// TIA Portal project "PRESS1-2-3" (V18)

(* hardware
DEVICE "S7-1200 station_1"  S7-1200 Station
   slot 0: "Rack_0"  S7-1200 Rack  Rack  V1.0
   slot 1: "PLC_1"  CPU 1212C DC/DC/DC  6ES7 212-1AE40-0XB0  V4.5
*)

// ===== PLC "PLC_1"  CPU 1212C DC/DC/DC =====

VAR_GLOBAL   // PLC tag table "Tabla de variables estándar"
   "Simulem 5V (24)" AT %Q0.0 : Bool;
   "Interruptor" AT %M50.0 : Bool;
   "Off_interruptor" AT %M50.1 : Bool;
   "System_Byte" AT %MB1 : Byte;
   "FirstScan" AT %M1.0 : Bool;
   "DiagStatusUpdate" AT %M1.1 : Bool;
   "AlwaysTRUE" AT %M1.2 : Bool;
   "AlwaysFALSE" AT %M1.3 : Bool;
   "System_Byte(1)" AT %MB1 : Byte;
   "Prensa_abaix" AT %I0.0 : Bool;
   "Prensa_dalt" AT %I0.1 : Bool;
   "Selector_Automatic" AT %I0.2 : Bool;
   "Sensor_mans" AT %I0.3 : Bool;
   "Maquina_endollada" AT %I0.4 : Bool;
END_VAR

VAR_GLOBAL   // PLC tag table "senyals_okuma"
   "nova_peca" AT %I0.7 : Bool;
   "servei" AT %I0.5 : Bool;
   "pedal" AT %I0.6 : Bool;
END_VAR

DATA_BLOCK "Prensa1"   // DB2
{ S7_Optimized_Access := 'FALSE' }
VERSION : 0.1
   VAR
      num_peces : UInt;
      temps_peca : Time;
      hora_peca : DTL;
      reset : UInt;
   END_VAR
BEGIN
END_DATA_BLOCK

DATA_BLOCK "vAR_Inpas"   // DB3
{ S7_Optimized_Access := 'FALSE' }
VERSION : 0.1
   VAR
      hora_actual : DTL;
      flanc2 : Bool;
      flanc1 : Bool;
      recompte_de_peces : Array[0..300] of Time;
   END_VAR
BEGIN
END_DATA_BLOCK

FUNCTION_BLOCK "Peca_acabada"   // FB1, LAD
TITLE = obtenim: temps de peça, hora inici, hora final
{ S7_Optimized_Access := 'TRUE' }
VERSION : 0.1
   VAR RETAIN
      OPC_Data : Struct
         Data_bool : Bool;
         Data_Int : Int;
         Data_String : String;
      END_STRUCT;
   END_VAR
   VAR_TEMP
      hora_actual : DTL;
      ok : Int;
   END_VAR
BEGIN

REGION Network 1: Obtenim la hora actual (hora de peça acabada)
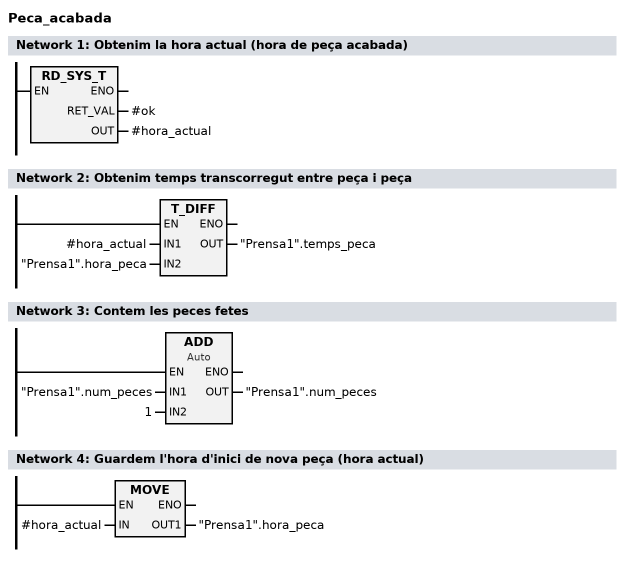
   #ok := RD_SYS_T(OUT => #hora_actual);
END_REGION

REGION Network 2: Obtenim temps transcorregut entre peça i peça
   "Prensa1".temps_peca := T_DIFF(IN1 := #hora_actual, IN2 := "Prensa1".hora_peca);
END_REGION

REGION Network 3: Contem les peces fetes
   RUNG wire#powerrail
      Add(in1 := "Prensa1".num_peces, in2 := 1, out => "Prensa1".num_peces)
   END_RUNG
   // the same network as SCL:
   "Prensa1".num_peces := "Prensa1".num_peces + 1;
END_REGION

REGION Network 4: Guardem l'hora d'inici de nova peça (hora actual)
   RUNG wire#powerrail
      Move(in := #hora_actual, out1 => "Prensa1".hora_peca)
   END_RUNG
   // the same network as SCL:
   "Prensa1".hora_peca := #hora_actual;
END_REGION
END_FUNCTION_BLOCK

FUNCTION "Peca_acabada_ok" : Void   // FC1, LAD
{ S7_Optimized_Access := 'TRUE' }
VERSION : 0.1
   VAR_INPUT
      hora_ultima_peca_in : DTL;
      num_peces_in : UInt;
   END_VAR
   VAR_OUTPUT
      hora_ultima_peca_out : DTL;
      temps_peca_out : Time;
      num_peces_out : UInt;
   END_VAR
   VAR_TEMP
      hora_actual : DTL;
      ok : Int;
   END_VAR
BEGIN

REGION Network 1: Obtenim la hora actual (hora de peça acabada)
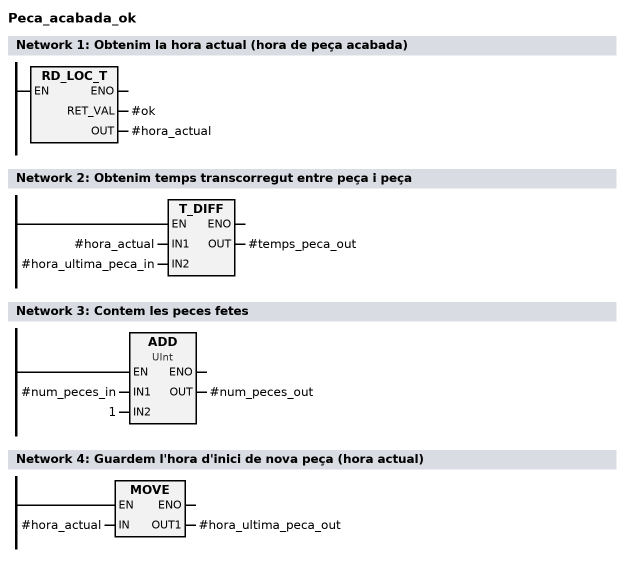
   #ok := RD_LOC_T(OUT => #hora_actual);
END_REGION

REGION Network 2: Obtenim temps transcorregut entre peça i peça
   #temps_peca_out := T_DIFF(IN1 := #hora_actual, IN2 := #hora_ultima_peca_in);
END_REGION

REGION Network 3: Contem les peces fetes
   RUNG wire#powerrail
      { S7_Templates := "SrcType := UInt" } Add(in1 := #num_peces_in, in2 := 1, out => #num_peces_out)
   END_RUNG
   // the same network as SCL:
   #num_peces_out := #num_peces_in + 1;
END_REGION

REGION Network 4: Guardem l'hora d'inici de nova peça (hora actual)
   RUNG wire#powerrail
      Move(in := #hora_actual, out1 => #hora_ultima_peca_out)
   END_RUNG
   // the same network as SCL:
   #hora_ultima_peca_out := #hora_actual;
END_REGION
END_FUNCTION

ORGANIZATION_BLOCK "Main"   // OB1, LAD, ProgramCycle
TITLE = "Main Program Sweep (Cycle)"
{ S7_Optimized_Access := 'TRUE' }
VERSION : 0.1
   VAR_INPUT
      Initial_Call : Bool;   // Initial call of this OB
      Remanence : Bool;   // =True, if remanent data are available
   END_VAR
   VAR_TEMP
      ok : Int;
      ok2 : Int;
   END_VAR
   VAR_TEMP   // added for the SCL form of the ladder/FBD networks
      _w1 : Bool;
   END_VAR
BEGIN

REGION Network 1: Detectar de peça finalitzada. Retorna temps i numero de la peça.
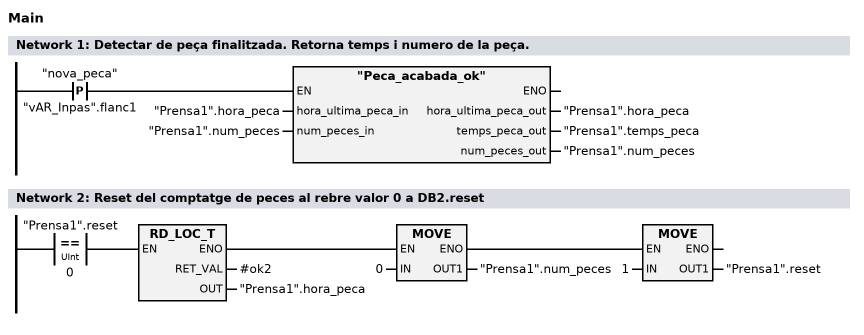
   RUNG wire#powerrail
      P_Contact(operand := "nova_peca", bit := "vAR_Inpas".flanc1)
      "Peca_acabada_ok"(hora_ultima_peca_in := "Prensa1".hora_peca, num_peces_in := "Prensa1".num_peces, hora_ultima_peca_out => "Prensa1".hora_peca, temps_peca_out => "Prensa1".temps_peca, num_peces_out => "Prensa1".num_peces)
   END_RUNG
   // the same network as SCL:
   #_w1 := "nova_peca" AND NOT "vAR_Inpas".flanc1;   // rising edge of "nova_peca"
   "vAR_Inpas".flanc1 := "nova_peca";
   IF #_w1 THEN
       "Peca_acabada_ok"(hora_ultima_peca_in := "Prensa1".hora_peca,
                         num_peces_in := "Prensa1".num_peces,
                         hora_ultima_peca_out => "Prensa1".hora_peca,
                         temps_peca_out => "Prensa1".temps_peca,
                         num_peces_out => "Prensa1".num_peces);
   END_IF;
END_REGION

REGION Network 2: Reset del comptatge de peces al rebre valor 0 a DB2.reset
   // ENO of a box is taken as its EN; it also drops when the box reports an error
   #_w1 := "Prensa1".reset = 0;
   IF #_w1 THEN
       #ok2 := RD_LOC_T(OUT => "Prensa1".hora_peca);
       "Prensa1".num_peces := 0;
       "Prensa1".reset := 1;
   END_IF;
END_REGION
END_ORGANIZATION_BLOCK

ORGANIZATION_BLOCK "Startup"   // OB100, LAD, Startup
TITLE = "Complete Restart"
{ S7_Optimized_Access := 'TRUE' }
VERSION : 0.1
   VAR_INPUT
      LostRetentive : Bool;   // True if retentive data are lost
      LostRTC : Bool;   // True if date and time are lost
   END_VAR
   VAR_TEMP
      ok : Int;
      ok2 : Int;
   END_VAR
BEGIN

REGION Network 1: Aquest bloc sempre em dona l'hora de l'any 1970...L'hora de system tambe dona 1970
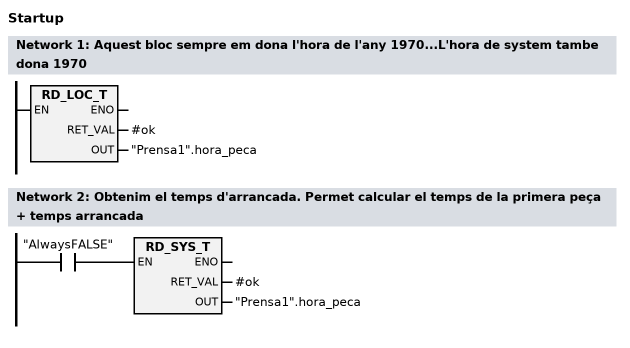
   #ok := RD_LOC_T(OUT => "Prensa1".hora_peca);
END_REGION

REGION Network 2: Obtenim el temps d'arrancada. Permet calcular el temps de la primera peça + temps arrancada
   IF "AlwaysFALSE" THEN #ok := RD_SYS_T(OUT => "Prensa1".hora_peca); END_IF;
END_REGION
END_ORGANIZATION_BLOCK